(* Schneider Machine Expert - Basic project VFD, file version 1.7.0.0 *)
(* ProjectInformations: Name=New project *)

HARDWARE
  Cpu 0: TM221ME32TK
  EthernetConfiguration: NetworkName=M221, IpAllocationMode=FixedAddress, IpAddress=0.0.0.0, SubnetMask=0.0.0.0
  SerialLineConfiguration: Baud=Baud19200, Parity=ParityEven, DataBits=DataBits8, StopBits=StopBits1, PhysicalMedium=PhysicalMediumRs485, TransmissionMode=TransmissionModeModbusRtu, SlaveId=1, Addressing=SlaveAddressing
  MastTask: UsePeriodScanMode=false, PeriodScan=100
  FastTask: Period=255
  CpuBehavior: StartingMode=StartAsPreviousState, AutoSaveRamOnEeprom=true, WatchdogPeriod=250

SYMBOLS  (address, symbol, comment, settings)
  %I0.0       "S1"
  %IW0.0      [Type=Type_0_10V, Scope=Scope_Normal, Minimum=0, Maximum=1000]

POU New POU
  (* SectionNumber=1 *)

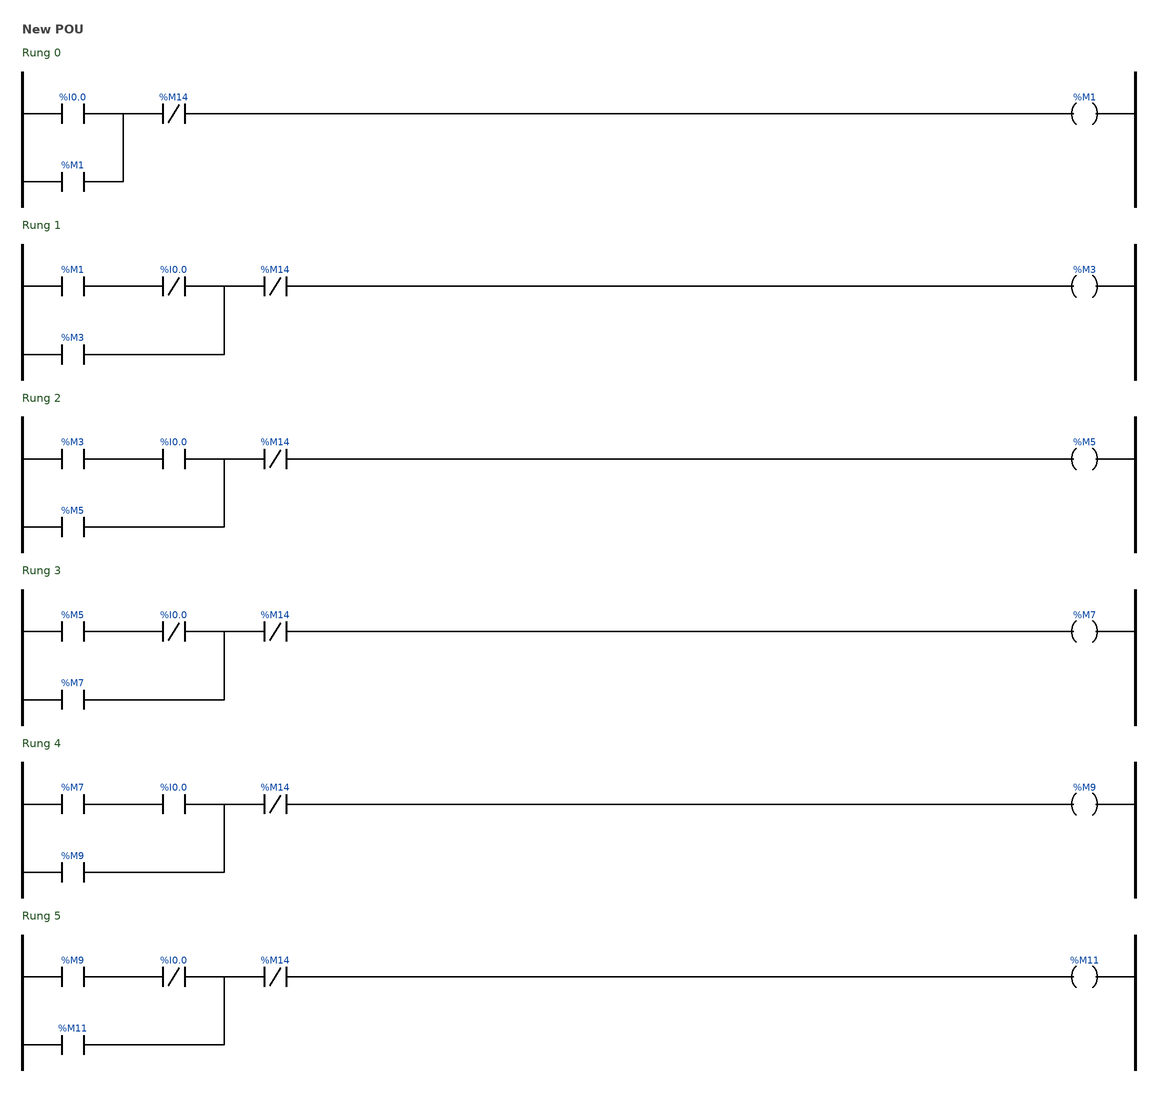

// Rung 0
  LD %I0.0
  OR %M1
  ANDN %M14
  ST %M1
  // as ST:
  //   %M1 := (%I0.0 OR %M1) AND NOT %M14;

// Rung 1
  LD %M1
  ANDN %I0.0
  OR %M3
  ANDN %M14
  ST %M3
  // as ST:
  //   %M3 := (%M1 AND NOT %I0.0 OR %M3) AND NOT %M14;

// Rung 2
  LD %M3
  AND %I0.0
  OR %M5
  ANDN %M14
  ST %M5
  // as ST:
  //   %M5 := (%M3 AND %I0.0 OR %M5) AND NOT %M14;

// Rung 3
  LD %M5
  ANDN %I0.0
  OR %M7
  ANDN %M14
  ST %M7
  // as ST:
  //   %M7 := (%M5 AND NOT %I0.0 OR %M7) AND NOT %M14;

// Rung 4
  LD %M7
  AND %I0.0
  OR %M9
  ANDN %M14
  ST %M9
  // as ST:
  //   %M9 := (%M7 AND %I0.0 OR %M9) AND NOT %M14;

// Rung 5
  LD %M9
  ANDN %I0.0
  OR %M11
  ANDN %M14
  ST %M11
  // as ST:
  //   %M11 := (%M9 AND NOT %I0.0 OR %M11) AND NOT %M14;

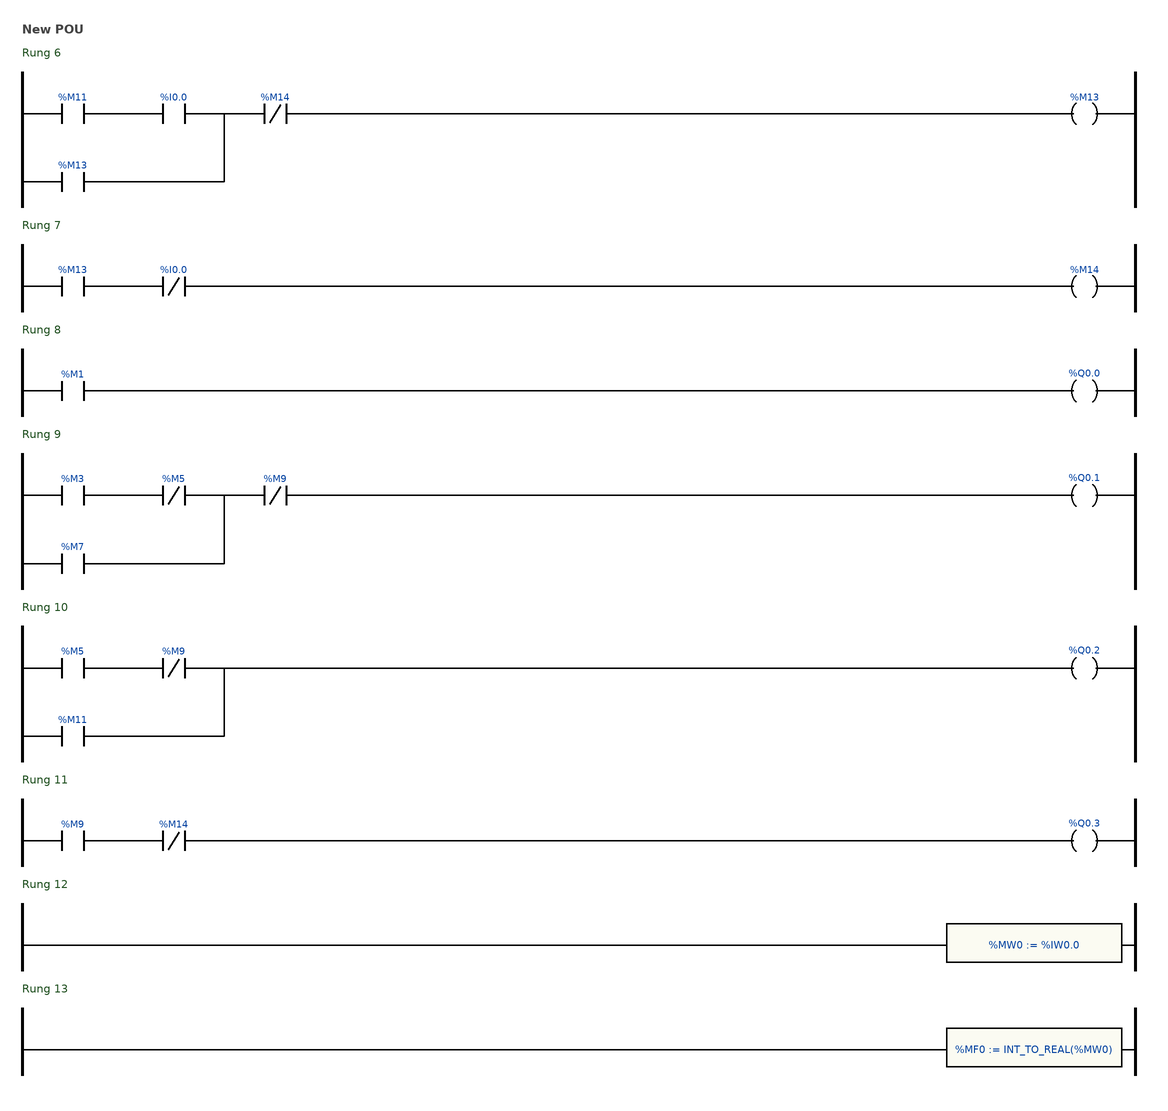

// Rung 6
  LD %M11
  AND %I0.0
  OR %M13
  ANDN %M14
  ST %M13
  // as ST:
  //   %M13 := (%M11 AND %I0.0 OR %M13) AND NOT %M14;

// Rung 7
  LD %M13
  ANDN %I0.0
  ST %M14
  // as ST:
  //   %M14 := %M13 AND NOT %I0.0;

// Rung 8
  LD %M1
  ST %Q0.0
  // as ST:
  //   %Q0.0 := %M1;

// Rung 9
  LD %M3
  ANDN %M5
  OR %M7
  ANDN %M9
  ST %Q0.1
  // as ST:
  //   %Q0.1 := (%M3 AND NOT %M5 OR %M7) AND NOT %M9;

// Rung 10
  LD %M5
  ANDN %M9
  OR %M11
  ST %Q0.2
  // as ST:
  //   %Q0.2 := %M5 AND NOT %M9 OR %M11;

// Rung 11
  LD %M9
  ANDN %M14
  ST %Q0.3
  // as ST:
  //   %Q0.3 := %M9 AND NOT %M14;

// Rung 12
  LD 1
  [ %MW0 := %IW0.0 ]
  // as ST:
  //   %MW0 := %IW0.0;

// Rung 13
  LD 1
  [ %MF0 := INT_TO_REAL ( %MW0 ) ]
  // as ST:
  //   %MF0 := INT_TO_REAL ( %MW0 );

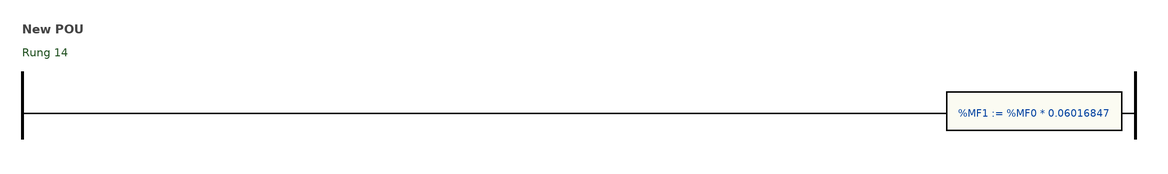

// Rung 14
  LD 1
  [ %MF1 := %MF0 * 0.06016847 ]
  // as ST:
  //   %MF1 := %MF0  *  0.06016847;
